FUNCTION SIND : LREAL
VAR_INPUT
	ANGLE:LREAL;
END_VAR
VAR
END_VAR

SIND:=SIN(DEG_TO_RAD(ANGLE));

END_FUNCTION

(* stored: Version 1.1.0.1, ProductVersion 3.1.4024.12
   POU SIND: Id {fb5e995e-4182-4df2-b1f8-e15d3e17d758}, SpecialFunc None *)
